// Mitsubishi GX Works2 project: group23_EX2   PLC: FX3G

// global labels: Global1
VAR_GLOBAL
  Start_Day AT X007 : BOOL;
  Emergency AT X005 : BOOL;
  work_day_light AT Y007 : BOOL;
  Stat_Melt AT X001 : BOOL;
  Start_Melt AT X001 : BOOL;
END_VAR
VAR_GLOBAL CONSTANT
  Chocolate_con : REAL := 400;
END_VAR
VAR_GLOBAL
  Chocolate_Light AT M1 : BOOL;
END_VAR
VAR_GLOBAL CONSTANT
  Nuts_con : REAL := 20.0;
END_VAR
VAR_GLOBAL
  Chocolate_Storge AT D1100 : REAL;
  Chocolate_Melt AT D2200 : REAL;
END_VAR
VAR_GLOBAL CONSTANT
  KKp : REAL := 400.0;
  Melt_Amount : REAL := 400.0;
END_VAR
VAR_GLOBAL
  Temp_Under45 AT X002 : BOOL;
  Melt_In_Process AT Y001 : BOOL;
  Melt_In_Proccess AT Y001 : BOOL;
END_VAR
VAR_GLOBAL CONSTANT
  Chocolate_min : REAL := 400;
END_VAR
VAR_GLOBAL
  Chocolate_low AT M1 : BOOL;
END_VAR
VAR_GLOBAL CONSTANT
  Nut_min : REAL := 100.0;
END_VAR
VAR_GLOBAL
  Nut_Storge AT D1200 : REAL;
  Nuts_low AT M2 : BOOL;
  Fistuk_Storge AT D1104 : REAL;
END_VAR
VAR_GLOBAL CONSTANT
  Fistuk_Min : REAL := 120.0;
END_VAR
VAR_GLOBAL
  Fistuk_low AT M3 : BOOL;
  Kadaif_Storge AT D1105 : REAL;
END_VAR
VAR_GLOBAL CONSTANT
  Kadaif_min : REAL := 60.0;
END_VAR
VAR_GLOBAL
  Kadif_low AT M4 : BOOL;
  Storage_Low AT M5 : BOOL;
  Chocolat_low AT M1 : BOOL;
  Start_Package AT Y001 : BOOL;
  Package_in_place AT X003 : BOOL;
  Melt_Finished AT M6 : BOOL;
  Move_chocolate AT M7 : BOOL;
  Chocolate_Mold AT D2100 : REAL;
  Melt_time AT TC1 : BOOL;
END_VAR
VAR_GLOBAL CONSTANT
  Melt_Constant : INT := 40;
END_VAR
VAR_GLOBAL
  Melt_time_TS AT TS1 : BOOL;
  Mold_in_proccess AT Y002 : BOOL;
  Input_Chocolate_strorge AT D1200 : REAL;
  Input_Nuts_strorge AT D1300 : REAL;
  Input_Nuts_strorage AT D1300 : REAL;
  Input_fistuk_storage AT D1400 : REAL;
  Input_kadaif_storage AT D1500 : REAL;
  Chocolate_storage AT D1600 : REAL;
  Nuts_storage AT D1700 : REAL;
  Fistuk_storage AT D1800 : REAL;
  Kadaif_storage AT D1900 : REAL;
  Mold_chocolate AT D2100 : REAL;
  Cream_fill AT X004 : BOOL;
  analog_input_1 AT D8280 : INT;
  Cream_type AT D2300 : INT;
  analog_light AT M8 : BOOL;
END_VAR
VAR_GLOBAL CONSTANT
  Con_2000 : INT := 2000;
END_VAR
VAR_GLOBAL
  Mix_nuts_cream_light AT M9 : BOOL;
  Dubai_cream_light AT M10 : BOOL;
  yuval AT Y004 : BOOL;
  Daniel AT Y005 : BOOL;
END_VAR
VAR_GLOBAL CONSTANT
  Con_K200 : INT := 2000;
  Con_K2000 : REAL := 2000;
END_VAR
VAR_GLOBAL
  Cream_type_INT AT D2200 : INT;
  Cream_type_Real AT D8000 : REAL;
END_VAR
VAR_GLOBAL CONSTANT
  Con_400 : REAL := 400.0;
  Con_5 : REAL := 5;
END_VAR
VAR_GLOBAL
  Cream_type_float AT D8000 : REAL;
  Flicker_light AT M9 : BOOL;
  M_10 AT M10 : BOOL;
  Flicker_time1 AT TC2 : BOOL;
  Flicker_time2 AT TC3 : BOOL;
END_VAR
VAR_GLOBAL CONSTANT
  flicker_const : INT := 20;
END_VAR
VAR_GLOBAL
  TS_2 AT TS2 : BOOL;
  TS_3 AT TS3 : BOOL;
  y_3 AT Y003 : BOOL;
  y_4 AT Y004 : BOOL;
  Flicker_time3 AT TC4 : BOOL;
END_VAR
VAR_GLOBAL CONSTANT
  Four_seconds : INT := 40;
END_VAR
VAR_GLOBAL
  TS_4 AT TS4 : BOOL;
END_VAR
VAR_GLOBAL CONSTANT
  Flicker_Constant : INT := 2;
  Four_second : INT := 40;
  Con100 : REAL := 100;
  Con20 : REAL := 20;
  Con120 : REAL := 120;
  Con60 : REAL := 60;
END_VAR
VAR_GLOBAL
  Start_cooling AT X006 : BOOL;
  Cool_time AT TC5 : BOOL;
END_VAR
VAR_GLOBAL CONSTANT
  Cooling_con : INT := 30;
END_VAR
VAR_GLOBAL
  TS_5 AT TS5 : BOOL;
  Y_6 AT Y006 : BOOL;
  Table_counter AT CC1 : BOOL;
  X_00 AT X000 : BOOL;
END_VAR
VAR_GLOBAL CONSTANT
  Con_4 : INT := 4;
END_VAR
VAR_GLOBAL
  Table_CS AT CS1 : BOOL;
  y_5 AT Y005 : BOOL;
END_VAR
VAR_GLOBAL CONSTANT
  Cons_4 : INT := 4;
  Const_4 : INT := 4;
  Con_1 : INT := 1;
  Const_four : INT := 4;
END_VAR
VAR_GLOBAL
  Table_counter1 AT CC1 : BOOL;
  CS_Table1 AT CS1 : BOOL;
END_VAR
VAR_GLOBAL CONSTANT
  Cons_10 : REAL := 10;
END_VAR
VAR_GLOBAL
  Num_Packages_Output : REAL;
  analog_output AT D8282 : INT;
  packages_num_output AT D8100 : REAL;
  packages_num_output1 AT D2100 : REAL;
  Chocolate_Melt_container AT D2700 : REAL;
END_VAR
VAR_GLOBAL CONSTANT
  Chocolate_container : REAL := 400;
END_VAR
VAR_GLOBAL
  Num_Packages1 AT D3000 : REAL;
  Input_Chocolate_strorage AT D1200 : REAL;
  packages_num_output2 AT D4000 : REAL;
END_VAR
VAR_GLOBAL CONSTANT
  Cons_400 : INT := 400;
  Cons_40 : INT := 40;
  Cons_5 : INT := 5;
  Five_second : INT := 50;
END_VAR

// task Task_01 (event TRUE, interval 0, priority 31): POU_01

PROGRAM POU_01
VAR CONSTANT
  Flicker_Con : INT := 2;
END_VAR
(* structured ladder/FBD written out as ST: instructions are called as NAME(EN, inputs, outputs); _pN, _eN, _tN stand for wires *)
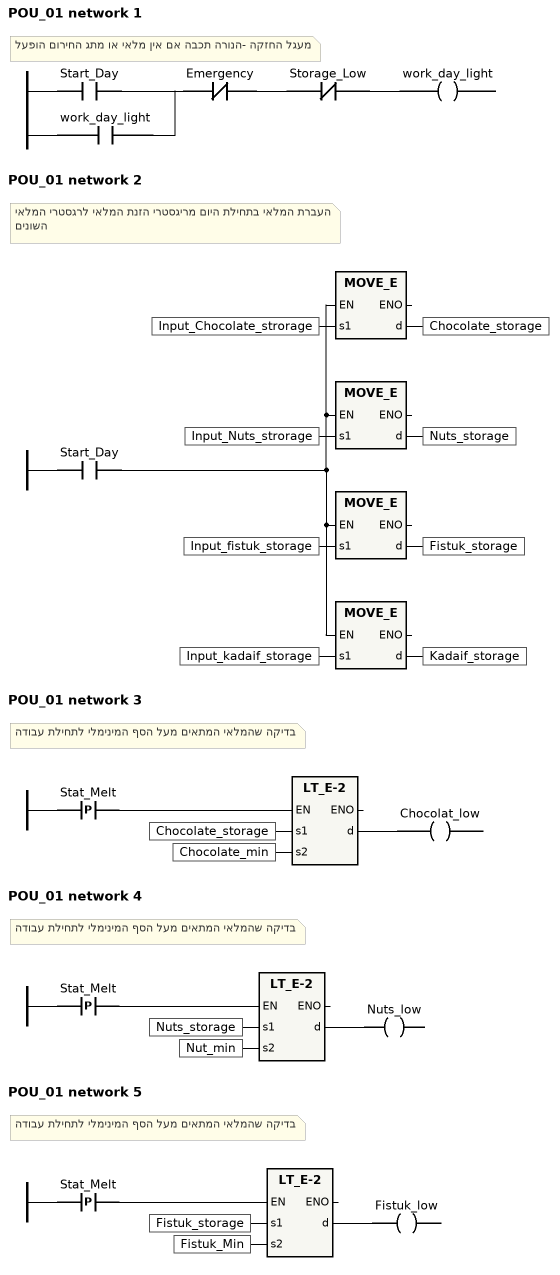
(* network 1 *)
(* מעגל החזקה -הנורה תכבה אם אין מלאי או מתג החירום הופעל *)
work_day_light := ((Start_Day OR work_day_light) AND NOT Emergency) AND NOT Storage_Low;
(* network 2 *)
(* העברת המלאי בתחילת היום מריגסטרי הזנת המלאי לרגסטרי המלאי השונים *)
MOVE_E(Start_Day, Input_Chocolate_strorage, Chocolate_storage);
MOVE_E(Start_Day, Input_Nuts_strorage, Nuts_storage);
MOVE_E(Start_Day, Input_fistuk_storage, Fistuk_storage);
MOVE_E(Start_Day, Input_kadaif_storage, Kadaif_storage);
(* network 3 *)
(* בדיקה שהמלאי המתאים מעל הסף המינימלי לתחילת עבודה *)
LT_E(LDP(TRUE, Stat_Melt), Chocolate_storage, Chocolate_min, _t1);
Chocolat_low := _t1;
(* network 4 *)
(* בדיקה שהמלאי המתאים מעל הסף המינימלי לתחילת עבודה *)
LT_E(LDP(TRUE, Stat_Melt), Nuts_storage, Nut_min, _t1);
Nuts_low := _t1;
(* network 5 *)
(* בדיקה שהמלאי המתאים מעל הסף המינימלי לתחילת עבודה *)
LT_E(LDP(TRUE, Stat_Melt), Fistuk_storage, Fistuk_Min, _t1);
Fistuk_low := _t1;
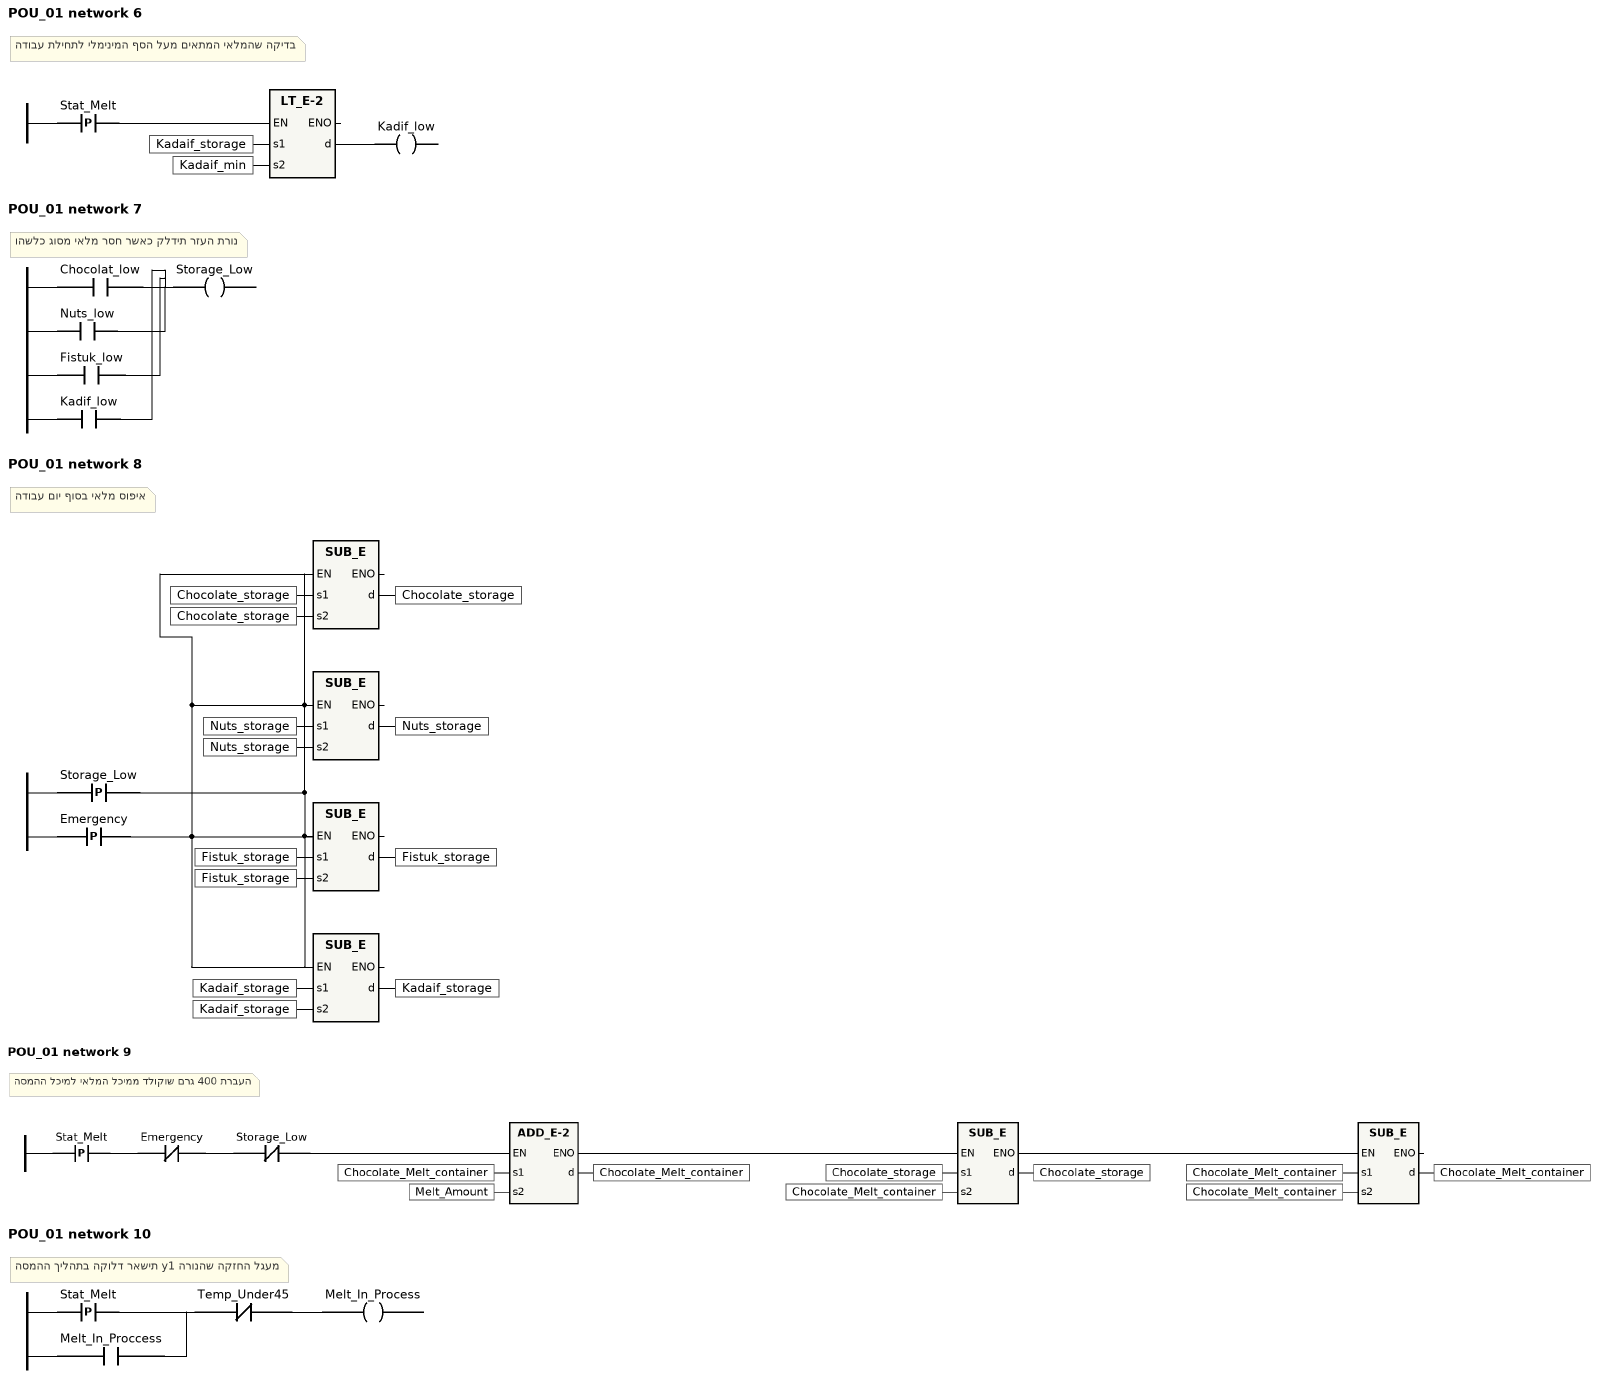
(* network 6 *)
(* בדיקה שהמלאי המתאים מעל הסף המינימלי לתחילת עבודה *)
LT_E(LDP(TRUE, Stat_Melt), Kadaif_storage, Kadaif_min, _t1);
Kadif_low := _t1;
(* network 7 *)
(* נורת העזר תידלק כאשר חסר מלאי מסוג כלשהו *)
Storage_Low := Chocolat_low OR Nuts_low OR Fistuk_low OR Kadif_low;
(* network 8 *)
(* איפוס מלאי בסוף יום עבודה *)
_p1 := LDP(TRUE, Storage_Low) OR LDP(TRUE, Emergency);
SUB_E(_p1, Chocolate_storage, Chocolate_storage, Chocolate_storage);
SUB_E(_p1, Nuts_storage, Nuts_storage, Nuts_storage);
SUB_E(_p1, Fistuk_storage, Fistuk_storage, Fistuk_storage);
SUB_E(_p1, Kadaif_storage, Kadaif_storage, Kadaif_storage);
(* network 9 *)
(* העברת 400 גרם שוקולד ממיכל המלאי למיכל ההמסה *)
_e1 := ADD_E(LDP(TRUE, Stat_Melt) AND NOT Emergency AND NOT Storage_Low, Chocolate_Melt_container, Melt_Amount, Chocolate_Melt_container);
_e2 := SUB_E(_e1, Chocolate_storage, Chocolate_Melt_container, Chocolate_storage);
SUB_E(_e2, Chocolate_Melt_container, Chocolate_Melt_container, Chocolate_Melt_container);
(* network 10 *)
(* מעגל החזקה שהנורה y1 תישאר דלוקה בתהליך ההמסה *)
Melt_In_Process := (LDP(TRUE, Stat_Melt) OR Melt_In_Proccess) AND NOT Temp_Under45;
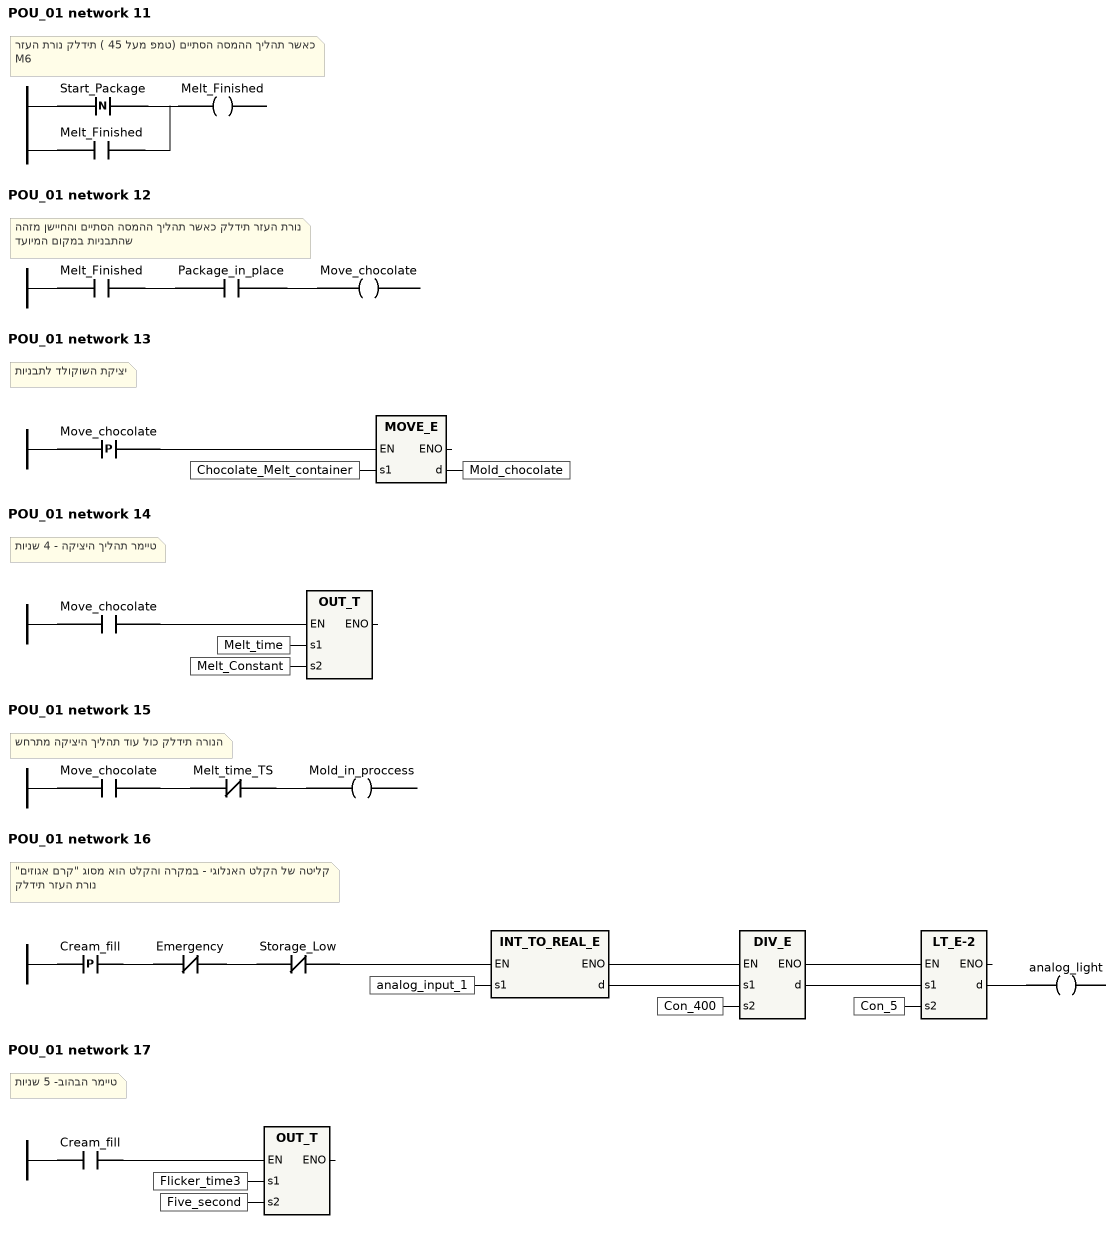
(* network 11 *)
(* כאשר תהליך ההמסה הסתיים (טמפ מעל 45 ) תידלק נורת העזר M6 *)
Melt_Finished := LDF(TRUE, Start_Package) OR Melt_Finished;
(* network 12 *)
(* נורת העזר תידלק כאשר תהליך ההמסה הסתיים והחיישן מזהה שהתבניות במקום המיועד *)
Move_chocolate := Melt_Finished AND Package_in_place;
(* network 13 *)
(* יציקת השוקולד לתבניות *)
MOVE_E(LDP(TRUE, Move_chocolate), Chocolate_Melt_container, Mold_chocolate);
(* network 14 *)
(* טיימר תהליך היציקה - 4 שניות *)
OUT_T(Move_chocolate, Melt_time, Melt_Constant);
(* network 15 *)
(* הנורה תידלק כול עוד תהליך היציקה מתרחש *)
Mold_in_proccess := Move_chocolate AND NOT Melt_time_TS;
(* network 16 *)
(* קליטה של הקלט האנלוגי - במקרה והקלט הוא מסוג "קרם אגוזים" נורת העזר תידלק *)
_e2 := INT_TO_REAL_E(LDP(TRUE, Cream_fill) AND NOT Emergency AND NOT Storage_Low, analog_input_1, _t1);
_e4 := DIV_E(_e2, _t1, Con_400, _t3);
LT_E(_e4, _t3, Con_5, _t5);
analog_light := _t5;
(* network 17 *)
(* טיימר הבהוב- 5 שניות *)
OUT_T(Cream_fill, Flicker_time3, Five_second);
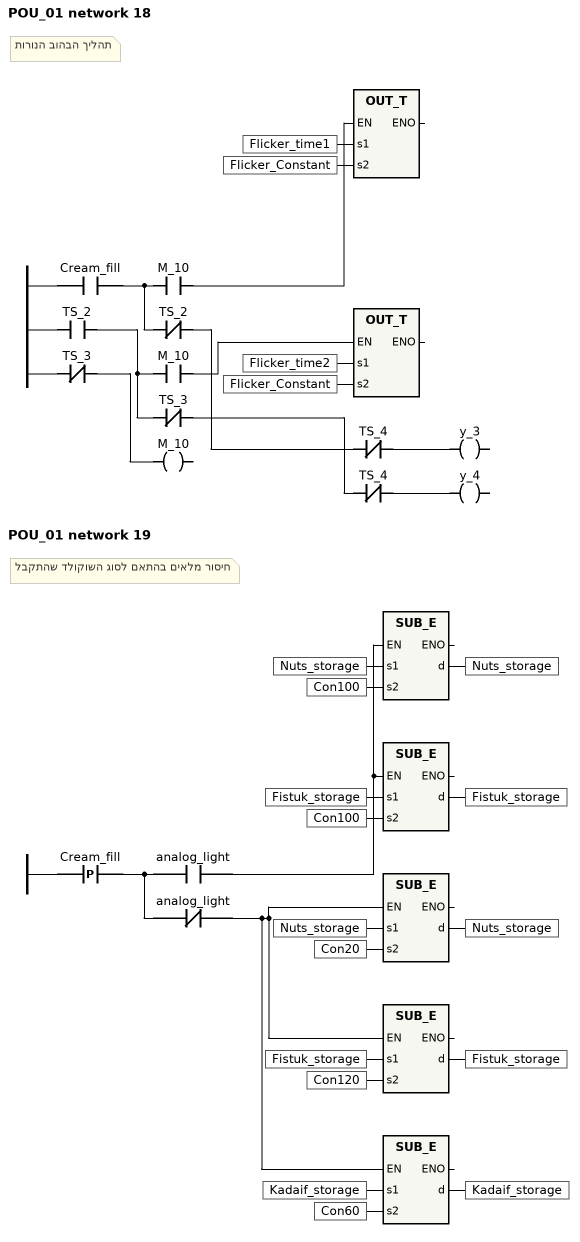
(* network 18 *)
(* תהליך הבהוב הנורות *)
OUT_T(Cream_fill AND M_10, Flicker_time1, Flicker_Constant);
y_3 := Cream_fill AND NOT TS_2 AND NOT TS_4;
OUT_T(TS_2 AND M_10, Flicker_time2, Flicker_Constant);
y_4 := TS_2 AND NOT TS_3 AND NOT TS_4;
M_10 := NOT TS_3;
(* network 19 *)
(* חיסור מלאים בהתאם לסוג השוקולד שהתקבל *)
_p1 := LDP(TRUE, Cream_fill);
_p2 := _p1 AND analog_light;
SUB_E(_p2, Nuts_storage, Con100, Nuts_storage);
SUB_E(_p2, Fistuk_storage, Con100, Fistuk_storage);
_p3 := _p1 AND NOT analog_light;
SUB_E(_p3, Nuts_storage, Con20, Nuts_storage);
SUB_E(_p3, Fistuk_storage, Con120, Fistuk_storage);
SUB_E(_p3, Kadaif_storage, Con60, Kadaif_storage);
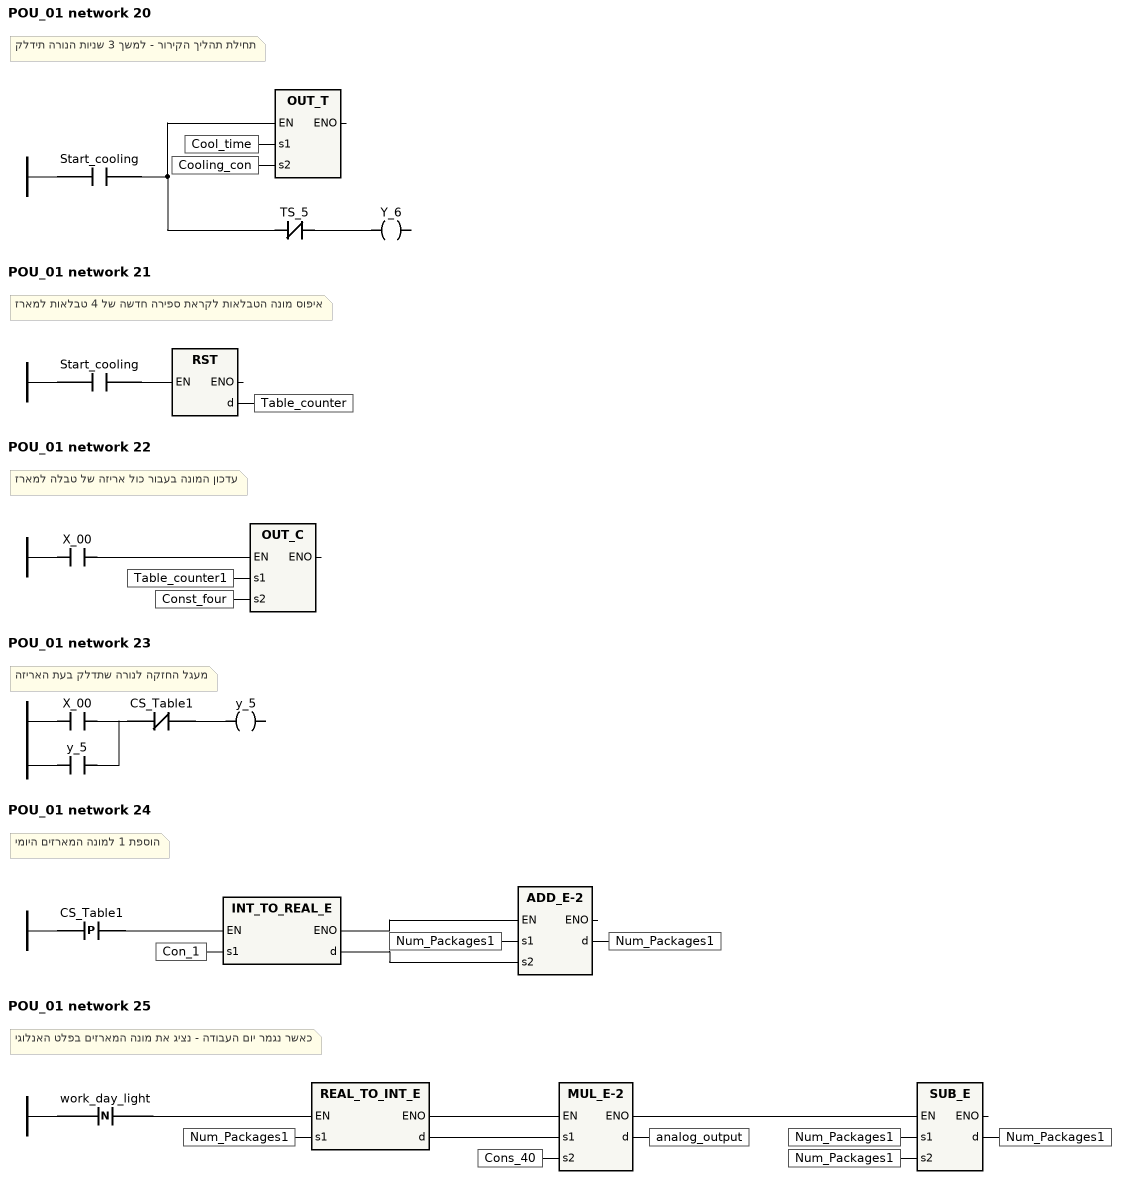
(* network 20 *)
(* תחילת תהליך הקירור - למשך 3 שניות הנורה תידלק *)
OUT_T(Start_cooling, Cool_time, Cooling_con);
Y_6 := Start_cooling AND NOT TS_5;
(* network 21 *)
(* איפוס מונה הטבלאות לקראת ספירה חדשה של 4 טבלאות למארז *)
RST(Start_cooling, Table_counter);
(* network 22 *)
(* עדכון המונה בעבור כול אריזה של טבלה למארז *)
OUT_C(X_00, Table_counter1, Const_four);
(* network 23 *)
(* מעגל החזקה לנורה שתדלק בעת האריזה *)
y_5 := (X_00 OR y_5) AND NOT CS_Table1;
(* network 24 *)
(* הוספת 1 למונה המארזים היומי *)
_e2 := INT_TO_REAL_E(LDP(TRUE, CS_Table1), Con_1, _t1);
ADD_E(_e2, Num_Packages1, _t1, Num_Packages1);
(* network 25 *)
(* כאשר נגמר יום העבודה - נציג את מונה המארזים בפלט האנלוגי *)
_e2 := REAL_TO_INT_E(LDF(TRUE, work_day_light), Num_Packages1, _t1);
_e3 := MUL_E(_e2, _t1, Cons_40, analog_output);
SUB_E(_e3, Num_Packages1, Num_Packages1, Num_Packages1);
END_PROGRAM
